(* LS Electric XG5000 project: project3 *)
(* PLC LSPLC *)

FUNCTION_BLOCK 위치사용
VAR_INPUT
    s11 : BOOL;
    s12 : BOOL;
    s13 : BOOL;
    s21 : BOOL;
    s22 : BOOL;
    s23 : BOOL;
    s31 : BOOL;
    s32 : BOOL;
    s33 : BOOL;
END_VAR
VAR_OUTPUT
    out11 : WORD;
    out12 : WORD;
    out13 : WORD;
    out21 : WORD;
    out22 : WORD;
    out23 : WORD;
    out31 : WORD;
    out32 : WORD;
    out33 : WORD;
END_VAR
VAR
    mout11 : INT;
    mout12 : INT;
    mout13 : INT;
    mout21 : INT;
    mout22 : INT;
    mout23 : INT;
    mout31 : INT;
    mout32 : INT;
    mout33 : INT;
END_VAR
VAR
    _e1 : R_TRIG;
    _e2 : F_TRIG;
    _e3 : R_TRIG;
    _e4 : F_TRIG;
    _e5 : R_TRIG;
    _e6 : F_TRIG;
    _e7 : R_TRIG;
    _e8 : F_TRIG;
    _e9 : R_TRIG;
    _e10 : F_TRIG;
    _e11 : R_TRIG;
    _e12 : F_TRIG;
    _e13 : R_TRIG;
    _e14 : F_TRIG;
    _e15 : R_TRIG;
    _e16 : F_TRIG;
    _e17 : R_TRIG;
    _e18 : F_TRIG;
END_VAR

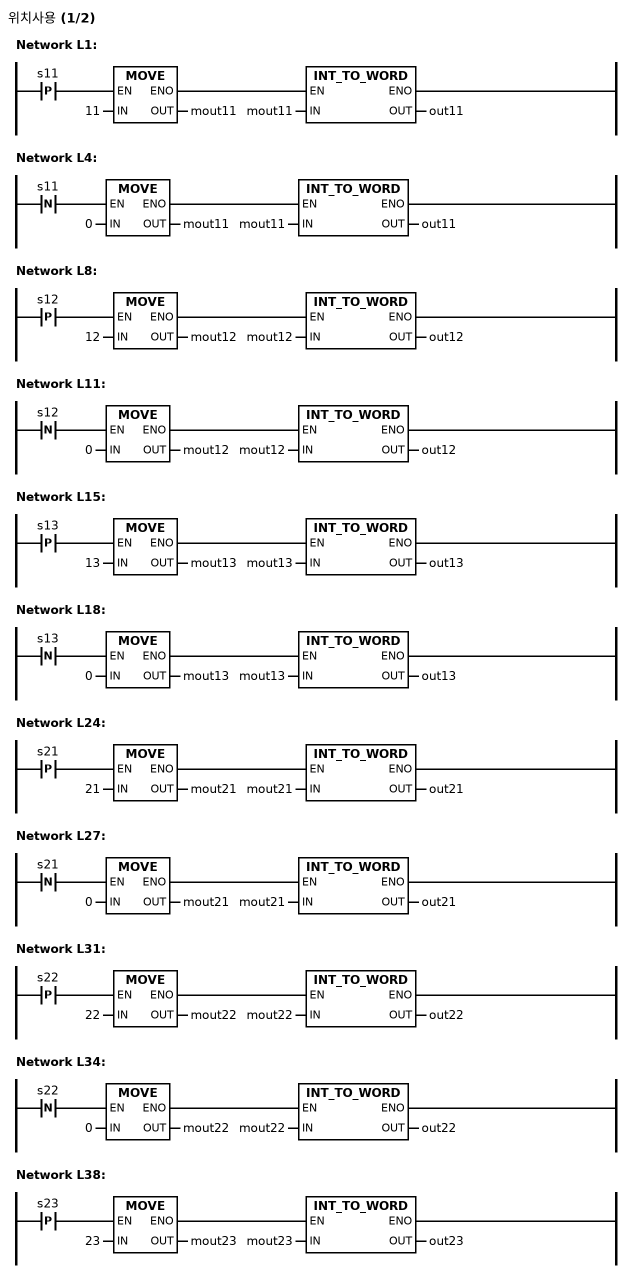
(* Rung L1 *)
_e1(CLK := s11);
IF _e1.Q THEN
    mout11 := 11;
    out11 := INT_TO_WORD(mout11);
END_IF;
(* Rung L4 *)
_e2(CLK := s11);
IF _e2.Q THEN
    mout11 := 0;
    out11 := INT_TO_WORD(mout11);
END_IF;
(* Rung L8 *)
_e3(CLK := s12);
IF _e3.Q THEN
    mout12 := 12;
    out12 := INT_TO_WORD(mout12);
END_IF;
(* Rung L11 *)
_e4(CLK := s12);
IF _e4.Q THEN
    mout12 := 0;
    out12 := INT_TO_WORD(mout12);
END_IF;
(* Rung L15 *)
_e5(CLK := s13);
IF _e5.Q THEN
    mout13 := 13;
    out13 := INT_TO_WORD(mout13);
END_IF;
(* Rung L18 *)
_e6(CLK := s13);
IF _e6.Q THEN
    mout13 := 0;
    out13 := INT_TO_WORD(mout13);
END_IF;
(* Rung L24 *)
_e7(CLK := s21);
IF _e7.Q THEN
    mout21 := 21;
    out21 := INT_TO_WORD(mout21);
END_IF;
(* Rung L27 *)
_e8(CLK := s21);
IF _e8.Q THEN
    mout21 := 0;
    out21 := INT_TO_WORD(mout21);
END_IF;
(* Rung L31 *)
_e9(CLK := s22);
IF _e9.Q THEN
    mout22 := 22;
    out22 := INT_TO_WORD(mout22);
END_IF;
(* Rung L34 *)
_e10(CLK := s22);
IF _e10.Q THEN
    mout22 := 0;
    out22 := INT_TO_WORD(mout22);
END_IF;
(* Rung L38 *)
_e11(CLK := s23);
IF _e11.Q THEN
    mout23 := 23;
    out23 := INT_TO_WORD(mout23);
END_IF;

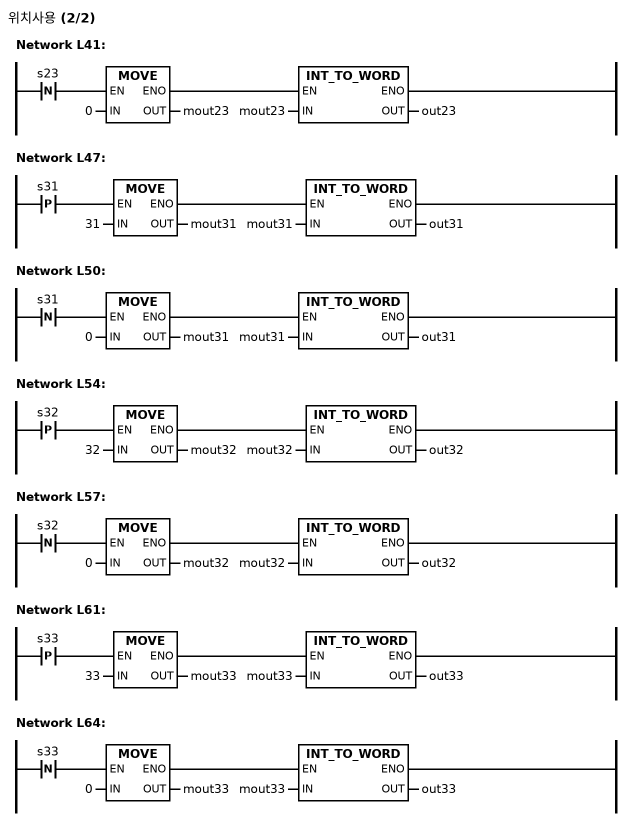
(* Rung L41 *)
_e12(CLK := s23);
IF _e12.Q THEN
    mout23 := 0;
    out23 := INT_TO_WORD(mout23);
END_IF;
(* Rung L47 *)
_e13(CLK := s31);
IF _e13.Q THEN
    mout31 := 31;
    out31 := INT_TO_WORD(mout31);
END_IF;
(* Rung L50 *)
_e14(CLK := s31);
IF _e14.Q THEN
    mout31 := 0;
    out31 := INT_TO_WORD(mout31);
END_IF;
(* Rung L54 *)
_e15(CLK := s32);
IF _e15.Q THEN
    mout32 := 32;
    out32 := INT_TO_WORD(mout32);
END_IF;
(* Rung L57 *)
_e16(CLK := s32);
IF _e16.Q THEN
    mout32 := 0;
    out32 := INT_TO_WORD(mout32);
END_IF;
(* Rung L61 *)
_e17(CLK := s33);
IF _e17.Q THEN
    mout33 := 33;
    out33 := INT_TO_WORD(mout33);
END_IF;
(* Rung L64 *)
_e18(CLK := s33);
IF _e18.Q THEN
    mout33 := 0;
    out33 := INT_TO_WORD(mout33);
END_IF;
END_FUNCTION_BLOCK

FUNCTION_BLOCK 초기화
VAR_INPUT
    초기화 : BOOL;
END_VAR
VAR_OUTPUT
    출력 : BOOL;
END_VAR
VAR
    INST1 : TON;
    INST2 : TP;
END_VAR

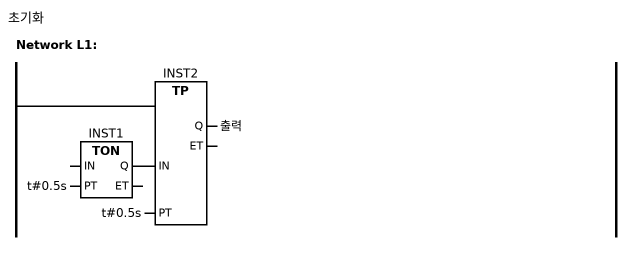
(* Rung L1 *)
INST1(IN := TRUE, PT := t#0.5s);
INST2(IN := INST1.Q, PT := t#0.5s, Q => 출력);
END_FUNCTION_BLOCK

FUNCTION_BLOCK move11
VAR_INPUT
    auto : BOOL;
END_VAR
VAR_OUTPUT
    move11 : BOOL; (* 11 *)
    move21 : BOOL; (* 21 *)
    move31 : BOOL; (* 31 *)
    move32 : BOOL; (* 32 *)
    move33 : BOOL; (* 33 *)
END_VAR
VAR
    X1 : TON;
    X2 : TON;
    X3 : TON;
    Y1 : TON;
    Y2 : TON;
END_VAR

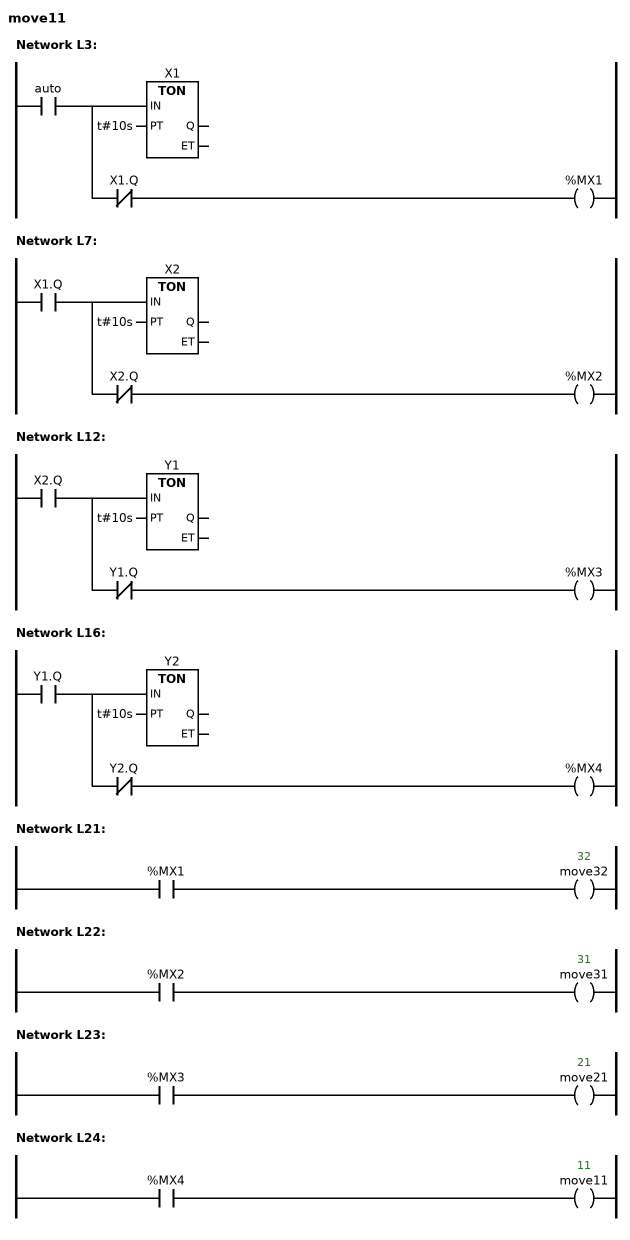
(* Rung L3 *)
X1(IN := auto, PT := t#10s);
%MX1 := auto AND NOT X1.Q;
(* Rung L7 *)
X2(IN := X1.Q, PT := t#10s);
%MX2 := X1.Q AND NOT X2.Q;
(* Rung L12 *)
Y1(IN := X2.Q, PT := t#10s);
%MX3 := X2.Q AND NOT Y1.Q;
(* Rung L16 *)
Y2(IN := Y1.Q, PT := t#10s);
%MX4 := Y1.Q AND NOT Y2.Q;
(* Rung L21 *)
move32 := %MX1;
(* Rung L22 *)
move31 := %MX2;
(* Rung L23 *)
move21 := %MX3;
(* Rung L24 *)
move11 := %MX4;
END_FUNCTION_BLOCK

FUNCTION_BLOCK move12
VAR_INPUT
    auto : BOOL;
END_VAR
VAR
    move12 : BOOL; (* 12 *)
    move22 : BOOL; (* 22 *)
    move32 : BOOL; (* 32 *)
    X1 : TON;
    X2 : TON;
    Y1 : TON;
    Y2 : TON;
END_VAR

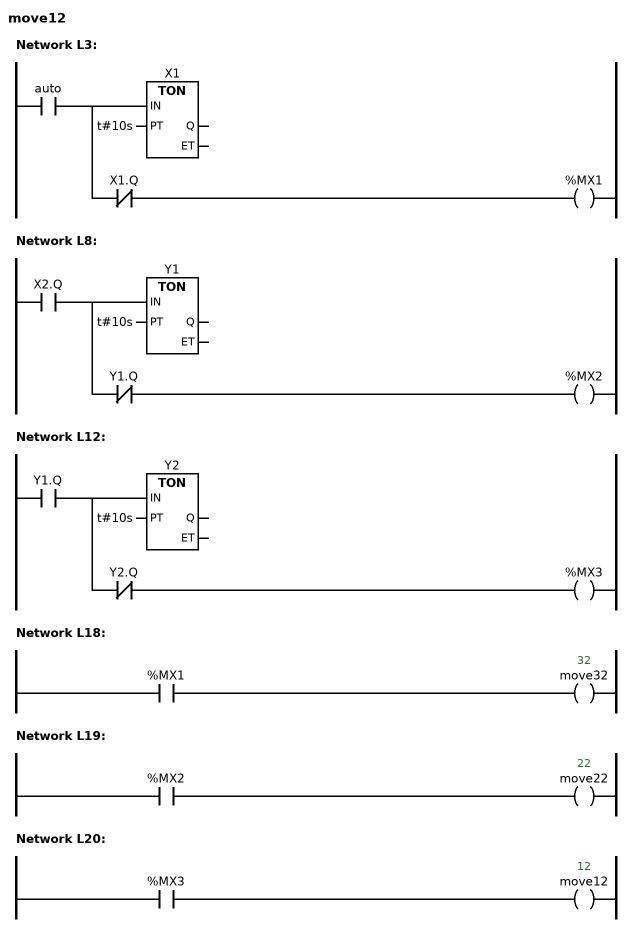
(* Rung L3 *)
X1(IN := auto, PT := t#10s);
%MX1 := auto AND NOT X1.Q;
(* Rung L8 *)
Y1(IN := X2.Q, PT := t#10s);
%MX2 := X2.Q AND NOT Y1.Q;
(* Rung L12 *)
Y2(IN := Y1.Q, PT := t#10s);
%MX3 := Y1.Q AND NOT Y2.Q;
(* Rung L18 *)
move32 := %MX1;
(* Rung L19 *)
move22 := %MX2;
(* Rung L20 *)
move12 := %MX3;
END_FUNCTION_BLOCK

FUNCTION_BLOCK move13
VAR_INPUT
    auto : BOOL;
END_VAR
VAR_OUTPUT
    move33 : BOOL; (* 33 *)
    move32 : BOOL; (* 32 *)
    move22 : BOOL;
    move12 : BOOL;
END_VAR
VAR
    move13 : BOOL; (* 13 *)
    move23 : BOOL; (* 23 *)
    X1 : TON;
    X2 : TON;
    Y1 : TON;
    Y2 : TON;
END_VAR

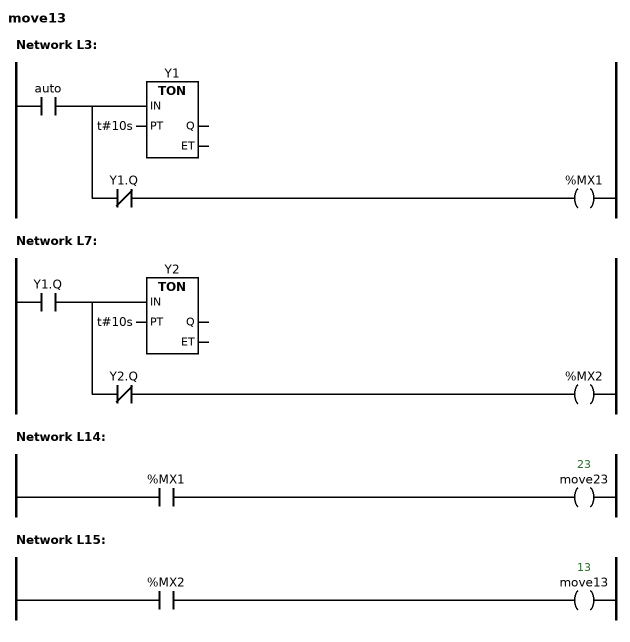
(* Rung L3 *)
Y1(IN := auto, PT := t#10s);
%MX1 := auto AND NOT Y1.Q;
(* Rung L7 *)
Y2(IN := Y1.Q, PT := t#10s);
%MX2 := Y1.Q AND NOT Y2.Q;
(* Rung L14 *)
move23 := %MX1;
(* Rung L15 *)
move13 := %MX2;
END_FUNCTION_BLOCK

PROGRAM NewProgram (* task: 스캔 프로그램 *)
VAR
    A AT %QX0.2.0 : BOOL;
    a1 : ARRAY[0..9] OF INT;
    AD : BOOL := 0;
    A_check AT %QX0.5.0 : BOOL;
    A_delay : TON;
    A_delay_유지 : BOOL;
    A_last : TON;
    A_pull : BOOL;
    A_push : BOOL;
    A_way AT %QX0.6.0 : BOOL;
    A단락 : BOOL;
    A센서 AT %QX0.9.0 : BOOL; (* 센서 *)
    A센서_딜레이 : TON;
    A센서상태변경 : TON;
    A센서지연 : TON;
    A센서지연1 : TON;
    A실린더_OFF AT %IX0.1.1 : BOOL; (* 실린더 *)
    A실린더_ON AT %IX0.1.0 : BOOL; (* 실린더 *)
    A지연 : TON;
    A차단 : TON;
    A카운트 : CTU_INT;
    A타이머 : TON;
    B AT %QX0.2.1 : BOOL;
    BD : BOOL := 0;
    B_check AT %QX0.5.1 : BOOL;
    B_delay : TON;
    B_delay_유지 : BOOL;
    B_last : TON;
    b_pull : BOOL;
    B_push : BOOL;
    B_way AT %QX0.6.1 : BOOL;
    B단락 : BOOL;
    B센서 AT %QX0.9.1 : BOOL; (* 센서 *)
    B센서_딜레이 : TON;
    B센서상태변경 : TON;
    B센서지연 : TON;
    B센서지연1 : TON;
    B실린더_OFF AT %IX0.1.3 : BOOL; (* 실린더 *)
    B실린더_ON AT %IX0.1.2 : BOOL; (* 실린더 *)
    B지연 : TON;
    B차단 : TON;
    B카운트 : CTU_INT;
    B타이머 : TON;
    C AT %QX0.2.2 : BOOL;
    CD : BOOL := 0;
    CU : BOOL;
    C_check AT %QX0.5.2 : BOOL;
    C_delay : TON;
    C_delay_유지 : BOOL;
    C_last : TON;
    c_out : BOOL;
    C_pull : BOOL;
    C_push : BOOL;
    C_way AT %QX0.6.2 : BOOL;
    C단락 : BOOL;
    C센서 AT %QX0.9.2 : BOOL; (* 센서 *)
    C센서_딜레이 : TON;
    C센서상태변경 : TON;
    C센서지연 : TON;
    C센서지연1 : TON;
    C실린더_OFF AT %IX0.1.5 : BOOL; (* 실린더 *)
    C실린더_ON AT %IX0.1.4 : BOOL; (* 실린더 *)
    C지연 : TON;
    C차단 : TON;
    C카운트 : CTUD_INT;
    C카운트1 : CTUD_INT;
    C타이머 : TON;
    C타이머1 : TON;
    C타이머2 : TON;
    D1 : WORD;
    D91 : TIME;
    delay : TP;
    done : BOOL;
    d_a AT %IW0.3.0 : WORD;
    d_a_out : UDINT;
    d_a_time : TIME;
    d_b AT %IW0.3.1 : WORD;
    d_b_out : UDINT;
    d_b_time : TIME;
    d_input : BOOL;
    fifo : FIFO_INT;
    INST : TP;
    LOAD : BOOL;
    OUT AT %QW0.8.0 : INT;
    prev AT %QW0.8.1 : WORD;
    prev_int : INT;
    rand : INT;
    reset : BOOL;
    RST : BOOL;
    s11 : BOOL;
    s12 : BOOL;
    s13 : BOOL;
    s21 : BOOL;
    s22 : BOOL;
    s23 : BOOL;
    s31 : BOOL;
    s32 : BOOL;
    s33 : BOOL;
    set : BOOL;
    signal : BOOL;
    stack : CTUD_INT;
    stack_max : INT := 9; (* max *)
    stack_센서 : BOOL;
    stack센서 : BOOL;
    start : BOOL;
    stop : BOOL;
    system_on AT %IX0.0.0 : BOOL;
    temp : BOOL;
    tepm : BOOL;
    test1 : BOOL;
    test2 : BOOL;
    three : WORD := 3;
    UNLD : BOOL;
    X1 : TON;
    X2 : TON;
    X3 : TON;
    Y1 : TON;
    Y2 : TON;
    Y3 : TON;
    _T15S : BOOL;
    긴급제동 : BOOL; (* RED *)
    난수1 : TON;
    난수2 : TON;
    난수회로차단 : TP;
    단선 AT %QX0.8.1 : BOOL;
    도착 AT %QX0.5.3 : BOOL;
    딜레이 : TON;
    랜덤수 : INT;
    명령 : BOOL;
    물품없음 : BOOL; (* WHITE *)
    백색등 : BOOL;
    선택값 : INT;
    수동 : BOOL;
    순환값 : WORD;
    숫자 : INT := 1;
    신호 AT %QX0.6.3 : BOOL;
    연기 : BOOL;
    위치사용 : 위치사용;
    임시 : BOOL;
    입력 : BOOL;
    입력1 AT %QX0.6.4 : BOOL;
    입력신호 AT %QW0.6.3 : INT;
    자동 : BOOL;
    저장 : FIFO_INT;
    정상가동 : BOOL; (* GREEN *)
    지연 : TON;
    지연1 : TP;
    초기화 : 초기화;
    출력 : BOOL;
    컨베이어벨트 AT %QX0.4.4 : BOOL;
    컨베이어타이머 : TON;
    하나출력 : BOOL;
END_VAR
VAR
    _t1 : BOOL;
    _e2 : R_TRIG;
    _e3 : F_TRIG;
    _e4 : F_TRIG;
    _e5 : F_TRIG;
    _e6 : F_TRIG;
    _e7 : R_TRIG;
    _e8 : R_TRIG;
    _p9 : BOOL;
    _p10 : BOOL;
    _e11 : R_TRIG;
    _p12 : BOOL;
    _p13 : BOOL;
    _e14 : R_TRIG;
    _p15 : BOOL;
    _p16 : BOOL;
END_VAR

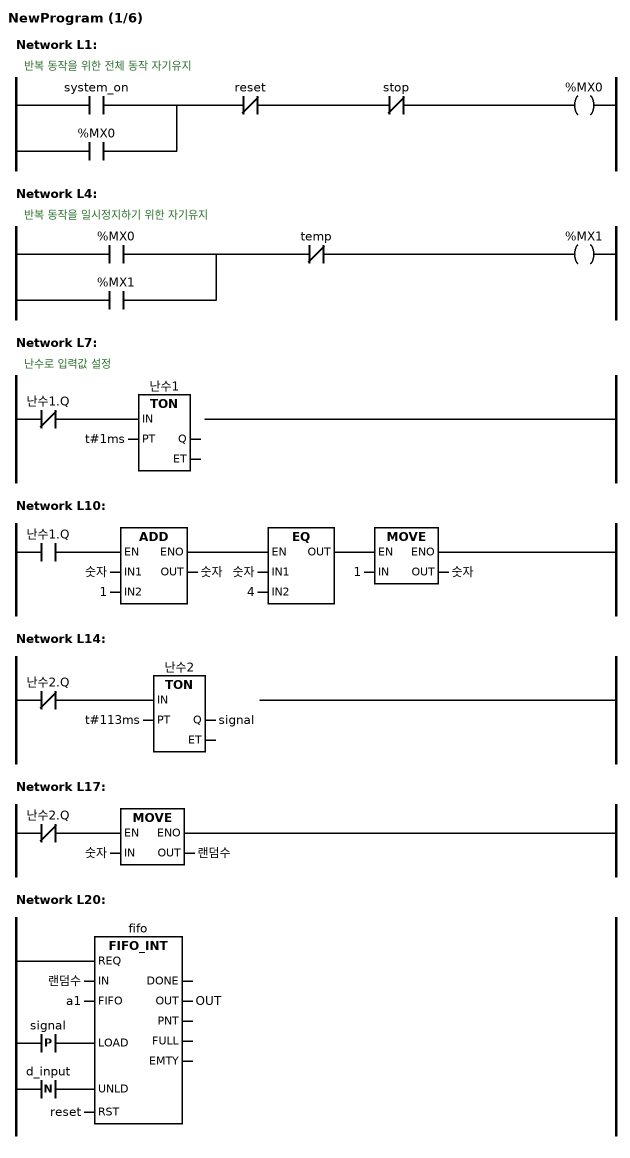
(* 반복 동작을 위한 전체 동작 자기유지 *)
(* Rung L1 *)
%MX0 := (system_on OR %MX0) AND NOT reset AND NOT stop;
(* 반복 동작을 일시정지하기 위한 자기유지 *)
(* Rung L4 *)
%MX1 := (%MX0 OR %MX1) AND NOT temp;
(* 난수로 입력값 설정 *)
(* Rung L7 *)
난수1(IN := NOT 난수1.Q, PT := t#1ms);
(* Rung L10 *)
IF 난수1.Q THEN
    숫자 := 숫자 + 1;
    _t1 := 숫자 = 4;
END_IF;
IF _t1 THEN 숫자 := 1; END_IF;
(* Rung L14 *)
난수2(IN := NOT 난수2.Q, PT := t#113ms, Q => signal);
(* Rung L17 *)
IF NOT 난수2.Q THEN 랜덤수 := 숫자; END_IF;
(* Rung L20 *)
_e2(CLK := signal);
_e3(CLK := d_input);
fifo(REQ := TRUE, IN := 랜덤수, FIFO := a1, LOAD := _e2.Q, UNLD := _e3.Q, RST := reset, OUT => OUT);

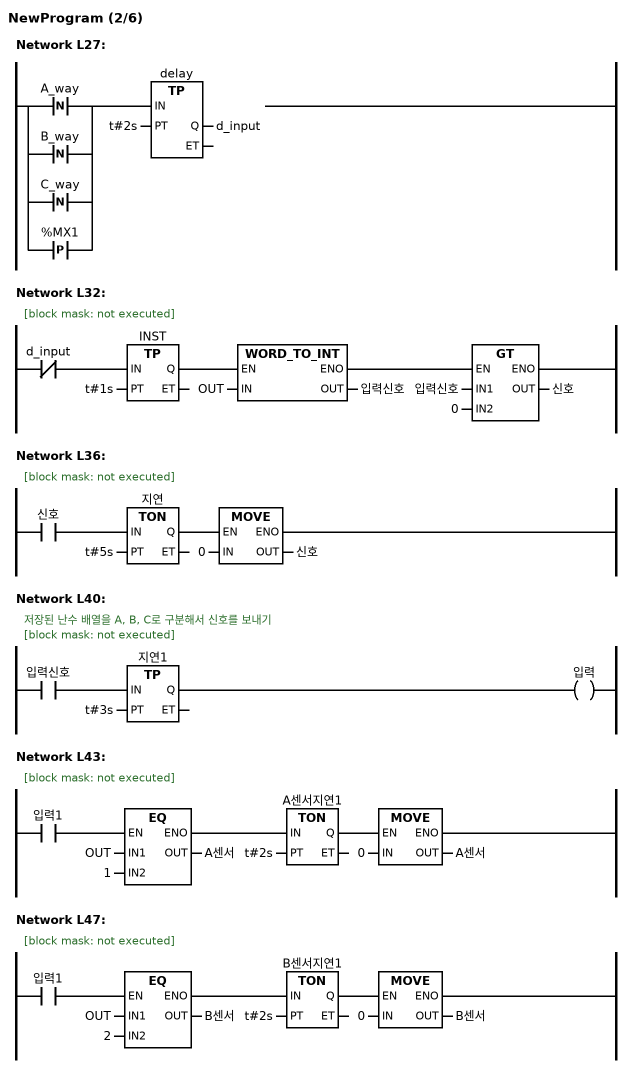
(* Rung L27 *)
_e4(CLK := A_way);
_e5(CLK := B_way);
_e6(CLK := C_way);
_e7(CLK := %MX1);
delay(IN := _e4.Q OR _e5.Q OR _e6.Q OR _e7.Q, PT := t#2s, Q => d_input);
(* Rung L32 is block-masked: not executed *)
// INST(IN := NOT d_input, PT := t#1s);
// IF INST.Q THEN
//     입력신호 := WORD_TO_INT(OUT);
//     신호 := 입력신호 > 0;
// END_IF;
(* Rung L36 is block-masked: not executed *)
// 지연(IN := 신호, PT := t#5s);
// IF 지연.Q THEN 신호 := 0; END_IF;
(* 저장된 난수 배열을 A, B, C로 구분해서 신호를 보내기 *)
(* Rung L40 is block-masked: not executed *)
// 지연1(IN := 입력신호, PT := t#3s);
// 입력 := 지연1.Q;
(* Rung L43 is block-masked: not executed *)
// IF 입력1 THEN A센서 := OUT = 1; END_IF;
// A센서지연1(IN := 입력1, PT := t#2s);
// IF A센서지연1.Q THEN A센서 := 0; END_IF;
(* Rung L47 is block-masked: not executed *)
// IF 입력1 THEN B센서 := OUT = 2; END_IF;
// B센서지연1(IN := 입력1, PT := t#2s);
// IF B센서지연1.Q THEN B센서 := 0; END_IF;

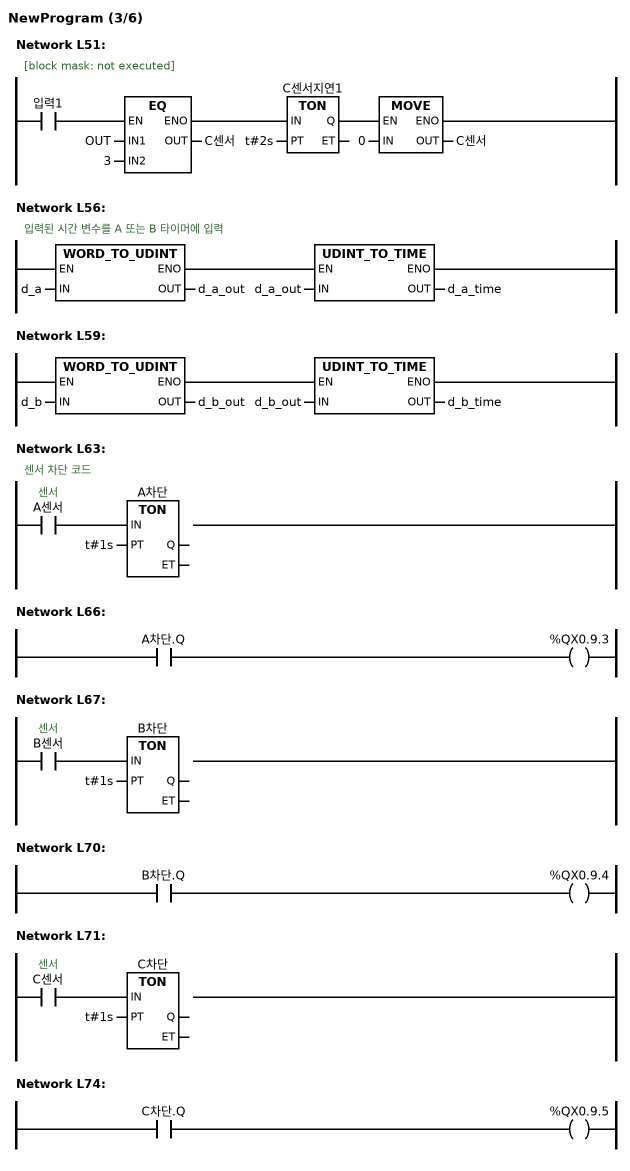
(* Rung L51 is block-masked: not executed *)
// IF 입력1 THEN C센서 := OUT = 3; END_IF;
// C센서지연1(IN := 입력1, PT := t#2s);
// IF C센서지연1.Q THEN C센서 := 0; END_IF;
(* 입력된 시간 변수를 A 또는 B 타이머에 입력 *)
(* Rung L56 *)
d_a_out := WORD_TO_UDINT(d_a);
d_a_time := UDINT_TO_TIME(d_a_out);
(* Rung L59 *)
d_b_out := WORD_TO_UDINT(d_b);
d_b_time := UDINT_TO_TIME(d_b_out);
(* 센서 차단 코드 *)
(* Rung L63 *)
A차단(IN := A센서, PT := t#1s);
(* Rung L66 *)
%QX0.9.3 := A차단.Q;
(* Rung L67 *)
B차단(IN := B센서, PT := t#1s);
(* Rung L70 *)
%QX0.9.4 := B차단.Q;
(* Rung L71 *)
C차단(IN := C센서, PT := t#1s);
(* Rung L74 *)
%QX0.9.5 := C차단.Q;

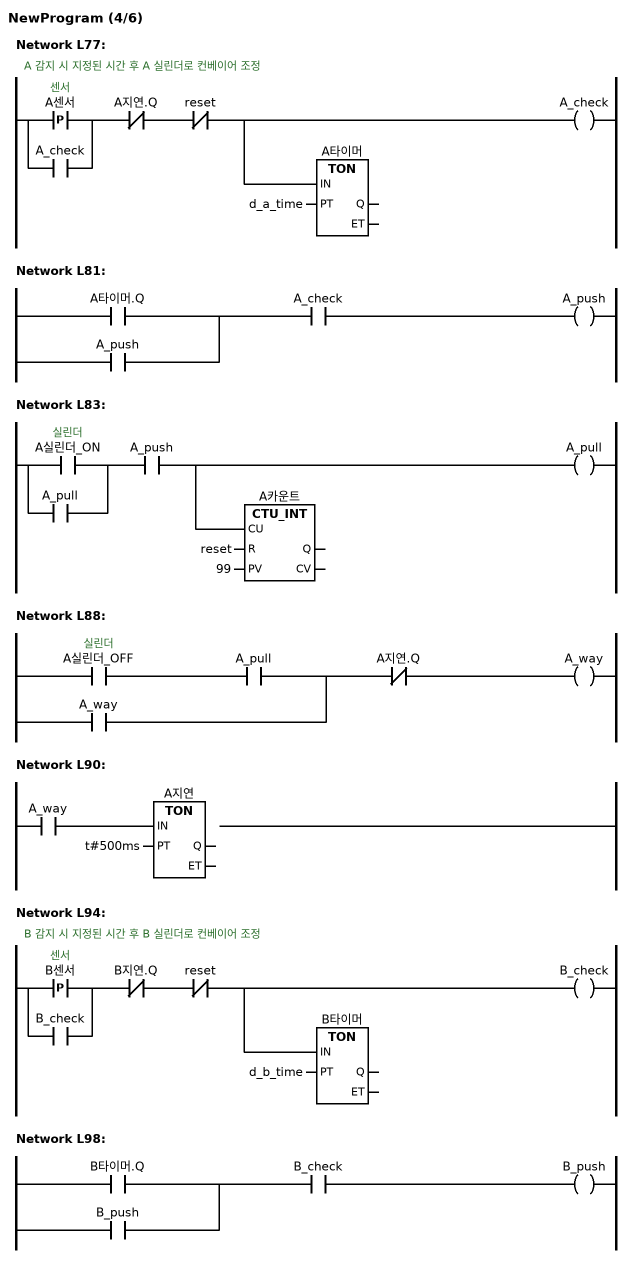
(* A 감지 시 지정된 시간 후 A 실린더로 컨베이어 조정 *)
(* Rung L77 *)
_e8(CLK := A센서);
_p9 := (_e8.Q OR A_check) AND NOT A지연.Q AND NOT reset;
A_check := _p9;
A타이머(IN := _p9, PT := d_a_time);
(* Rung L81 *)
A_push := (A타이머.Q OR A_push) AND A_check;
(* Rung L83 *)
_p10 := (A실린더_ON OR A_pull) AND A_push;
A_pull := _p10;
A카운트(CU := _p10, R := reset, PV := 99);
(* Rung L88 *)
A_way := ((A실린더_OFF AND A_pull) OR A_way) AND NOT A지연.Q;
(* Rung L90 *)
A지연(IN := A_way, PT := t#500ms);
(* B 감지 시 지정된 시간 후 B 실린더로 컨베이어 조정 *)
(* Rung L94 *)
_e11(CLK := B센서);
_p12 := (_e11.Q OR B_check) AND NOT B지연.Q AND NOT reset;
B_check := _p12;
B타이머(IN := _p12, PT := d_b_time);
(* Rung L98 *)
B_push := (B타이머.Q OR B_push) AND B_check;

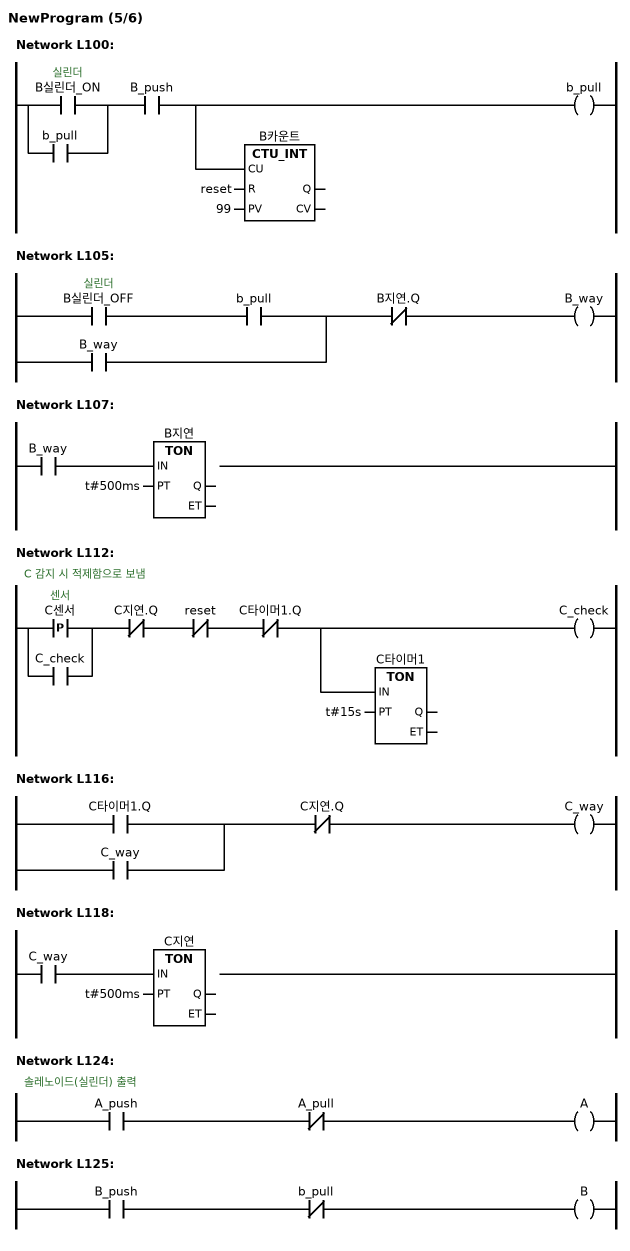
(* Rung L100 *)
_p13 := (B실린더_ON OR b_pull) AND B_push;
b_pull := _p13;
B카운트(CU := _p13, R := reset, PV := 99);
(* Rung L105 *)
B_way := ((B실린더_OFF AND b_pull) OR B_way) AND NOT B지연.Q;
(* Rung L107 *)
B지연(IN := B_way, PT := t#500ms);
(* C 감지 시 적제함으로 보냄 *)
(* Rung L112 *)
_e14(CLK := C센서);
_p15 := (_e14.Q OR C_check) AND NOT C지연.Q AND NOT reset AND NOT C타이머1.Q;
C_check := _p15;
C타이머1(IN := _p15, PT := t#15s);
(* Rung L116 *)
C_way := (C타이머1.Q OR C_way) AND NOT C지연.Q;
(* Rung L118 *)
C지연(IN := C_way, PT := t#500ms);
(* 솔레노이드(실린더) 출력 *)
(* Rung L124 *)
A := A_push AND NOT A_pull;
(* Rung L125 *)
B := B_push AND NOT b_pull;

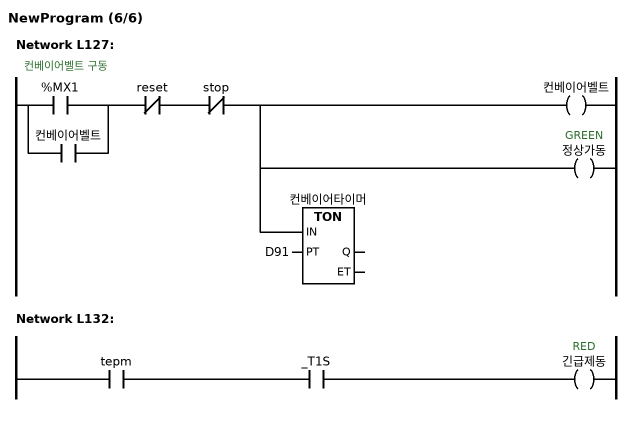
(* 컨베이어벨트 구동 *)
(* Rung L127 *)
_p16 := (%MX1 OR 컨베이어벨트) AND NOT reset AND NOT stop;
컨베이어벨트 := _p16;
정상가동 := _p16;
컨베이어타이머(IN := _p16, PT := D91);
(* Rung L132 *)
긴급제동 := tepm AND _T1S;
END_PROGRAM